FUNCTION_BLOCK F_UINT_TO_BOOL (* Service Interface Function Block Type *)
  (* Standard: 61499-2 *)
  (* Version 0.0, 2013-04-15, 4DIAC-IDE, 4DIAC-Consortium *)
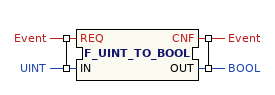
  EVENT_INPUT
    REQ WITH IN; (* Service Request *)
  END_EVENT
  EVENT_OUTPUT
    CNF WITH OUT; (* Confirmation of Requested Service *)
  END_EVENT
  VAR_INPUT
    IN : UINT; (* input value *)
  END_VAR
  VAR_OUTPUT
    OUT : BOOL; (* output value *)
  END_VAR
  (* Service APPLICATION/RESOURCE: Service Interface Function Block Type *)
END_FUNCTION_BLOCK
